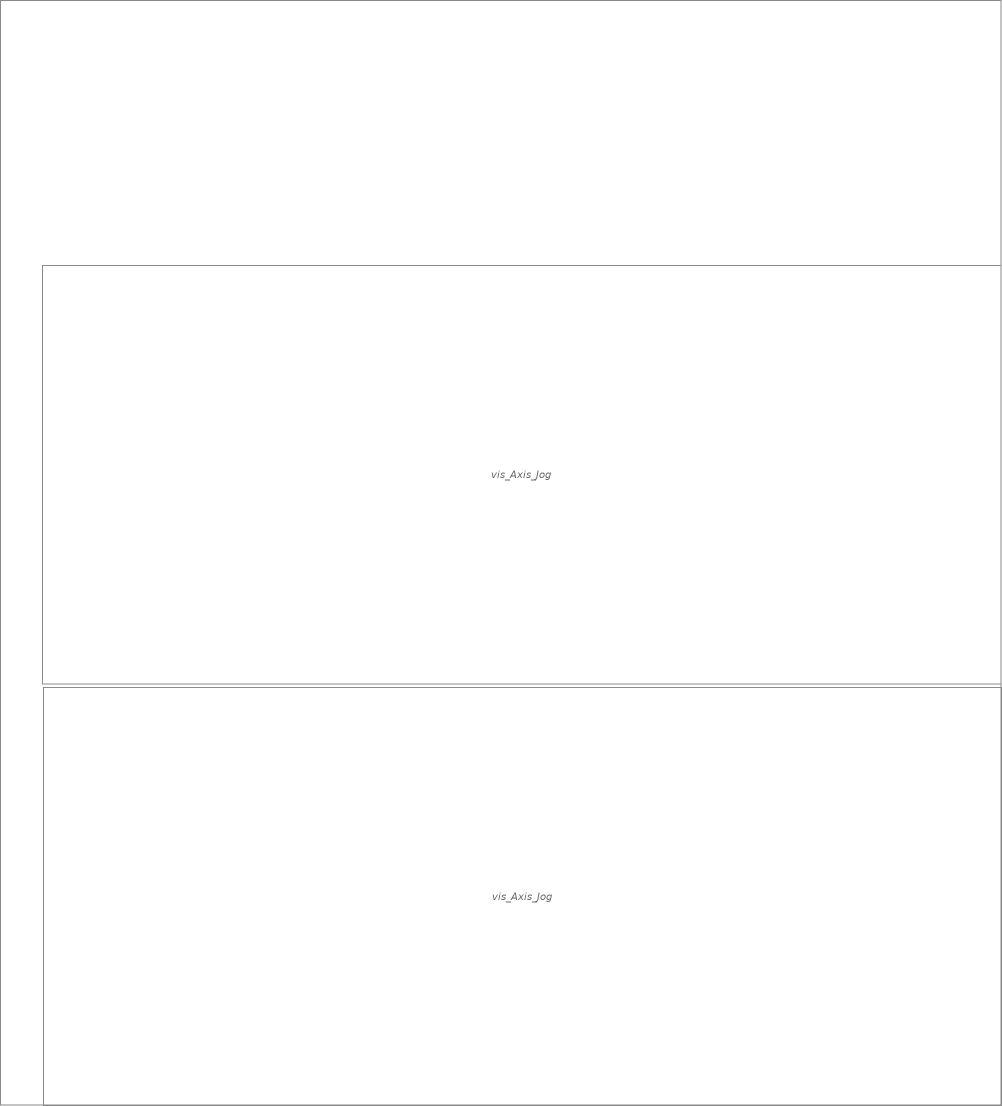
VISUALIZATION vis_Axis  // 1002x1106
    Frame (42,265 959x419)
        shows vis_Axis_Jog(Axis := stAxis[1])
    Frame (43,687 959x419)
        shows vis_Axis_Jog(Axis := stAxis[2])
END_VISUALIZATION

(* stored: Version 1.1.0.1, ProductVersion 3.1.4024.12
   Visu vis_Axis: Id {995578a7-d7aa-4a62-af70-88459ac04320} *)
